{attribute 'qualified_only'}
{attribute 'strict'}
TYPE SwitchState :
(
	Up := 0,
	Middle := 1,
	Down := 2,
	Moving := 3
);
END_TYPE

(* stored: Version 1.1.0.1, ProductVersion 3.1.4024.11
   DUT SwitchState: Id {a09ec9dc-21a0-403a-8bcf-f89326fb2f3c} *)
